FUNCTION_BLOCK FB_Logger
VAR_INPUT
	i_CloseSocket	:	BOOL := FALSE;
	i_bReset		:	BOOL := FALSE;
END_VAR
VAR
	fbUDPSocketManager	:	FB_ConnectionlessSocket;
	udpSocket			:	T_HSOCKET;
	fbUDPSocketSend		:	FB_SocketUdpSendTo;
	sOutgoingMesg		:	T_MaxString;
	eState				:	E_MessengerState;
	stDiag				:	ST_fbDiagnostics;
	rtReset				:	R_TRIG;
	fbGetSystemTime		:	FB_LocalSystemTime := (bEnable := TRUE);
	fbGetHostName		:	FB_GetHostName := (bExecute := TRUE, sNetID := '');
	ctuSentSomething	:	CTU := (PV := 100);
	rtSocketSendErr		:	R_TRIG;
END_VAR
VAR CONSTANT

END_VAR

(* Syslog Logger
A. Wallace 2016-9-3

This is used to pass PLC notification messeges to a syslog server.

This POU constantly attempts to send out messages from the global buffer.
*)

gfbBuffer.pBuffer := ADR(gMesgBuffer); 
gfbBuffer.cbBuffer:= SIZEOF(gMesgBuffer);

fbGetSystemTime(); 
IF fbGetSystemTime.bValid THEN
	gsCurrentTime := SYSTEM_TIME_TO_RFC3339(fbGetSystemTime.systemTime);
ELSE
	gsCurrentTime := cNILVALUE;
END_IF

fbGetHostName();
IF NOT (fbGetHostName.bBusy OR fbGetHostName.bError) THEN
	gsHostName := fbGetHostName.sHostName;
ELSE
	gsHostName := cNILVALUE;
END_IF

IF i_CloseSocket THEN 
	eState := E_MessengerState.CloseSocket; 
END_IF

rtReset(CLK:=i_bReset);
IF rtReset.Q THEN
	eState := E_MessengerState.CreateSocket;
	i_bReset R= i_bReset;
END_IF

rtSocketSendErr(CLK:=fbUDPSocketSend.bError);

CASE eState OF
	E_MessengerState.Init:
		;
	E_MessengerState.CreateSocket:
		fbUDPSocketManager.nLocalPort := g_udpSyslog;
		fbUDPSocketManager.bEnable := TRUE;
		
		IF fbUDPSocketManager.eState = E_SocketConnectionlessState.eSOCKET_CREATED THEN
			eState := E_MessengerState.Active;
		ELSIF fbUDPSocketManager.bError THEN
			eState := E_MessengerState.Err;
			fbUDPSocketManager.bEnable := FALSE;
			stDiag.fString( sOut=>stDiag.asResults[stDiag.resultIdx.IncVal()], sFormat:='Socketmanger error in createsocket: %d', arg1:=F_UDINT(fbUDPSocketManager.nErrID));
		//ELSE
			//eState := Err;
			//stDiag.fString( sOut=>stDiag.asResults[stDiag.resultIdx.IncVal()], sFormat:='Something else happened in createsocket -> error');
		END_IF
	E_MessengerState.Active:
		IF fbUDPSocketManager.eState = E_SocketConnectionlessState.eSOCKET_TRANSIENT  OR 
			fbUDPSocketManager.bError THEN
			eState := E_MessengerState.Err; 
			stDiag.fString( sOut=>stDiag.asResults[stDiag.resultIdx.IncVal()], sFormat:='Socketmanager error in active: %d', arg1:=F_UDINT(fbUDPSocketManager.nErrId));
		END_IF
		
		// While the socket is active, go ahead and send whatever is in the buffer
		IF rtSocketSendErr.Q THEN
			eState := E_MessengerState.Err;
			stDiag.fString( sOut=>stDiag.asResults[stDiag.resultIdx.IncVal()], sFormat:='Socket send error: %d', arg1:=F_UDINT(fbUDPSocketSend.nErrId));
		ELSIF gfbBuffer.nCount > 0 AND NOT fbUDPSocketSend.bBusy THEN
			gfbBuffer.A_RemoveHead(getValue=>sOutgoingMesg);
			fbUDPSocketSend.bExecute := TRUE; //reset in the action after busy goes true
			IF sOutgoingMesg <> '' THEN
				ctuSentSomething(CU:=TRUE);
			END_IF
		ELSIF gfbBuffer.nCount = 0 OR fbUDPSocketSend.bBusy THEN
			stDiag.fString( sOut=>stDiag.asResults[stDiag.resultIdx.IncVal()], sFormat:='Waiting to send');
			ctuSentSomething(CU:=FALSE);
		ELSE
			eState := E_MessengerState.Err;
			stDiag.fString( sOut=>stDiag.asResults[stDiag.resultIdx.IncVal()], sFormat:='Something else happened in active -> error');
		END_IF
		
	E_MessengerState.CloseSocket:
		fbUDPSocketManager.bEnable R= i_CloseSocket;
		IF fbUDPSocketManager.eState = E_SocketConnectionlessState.eSOCKET_CLOSED THEN
			eState := E_MessengerState.Init;
		ELSIF fbUDPSocketManager.bBusy AND NOT fbUDPSocketManager.bEnable THEN
			;
		ELSIF fbUDPSocketManager.bError THEN
			eState := E_MessengerState.Err;
		ELSE
			eState := E_MessengerState.Err;
		END_IF
	E_MessengerState.Err:
		eState := E_MessengerState.Init;
		stDiag.asResults[stDiag.resultIdx.IncVal()] := 'Moving back to Init state from Error';
END_CASE



Manager();
SocketSendTo();

ACTION Manager:
fbUDPSocketManager(hSocket => udpSocket);
END_ACTION

ACTION SocketSendTo:
fbUDPSocketSend.hSocket := udpSocket;
fbUDPSocketSend.sRemoteHost := g_psLogHost;
fbUDPSocketSend.nRemotePort := g_udpSyslog;
fbUDPSocketSend.pSrc := ADR(sOutgoingMesg);
fbUDPSocketSend.cbLen := SIZEOF(sOutgoingMesg);
fbUDPSocketSend();
fbUDPSocketSend.bExecute R= fbUDPSocketSend.bBusy;
END_ACTION

END_FUNCTION_BLOCK

(* stored: Version 1.1.0.1, ProductVersion 3.1.4022.10
   POU FB_Logger: Id {227c1bce-209d-4aad-8160-124282bb6370}, SpecialFunc None
   Action Manager: Id {0b30d4fb-bcf3-449a-83ce-64e06542700f}
   Action SocketSendTo: Id {fca34bf9-1619-4cff-a5ea-95f906bcb6c8} *)
